// TIA Portal V19 export
DATA_BLOCK "DB_Prog_edit"   // DB800
{ S7_Optimized_Access := 'FALSE' }
// stored: AutoNumber false
   VAR RETAIN
      akt_edit_prog : Int;
      akt_Aufgabe_Prog : Int;
      old_Aufgabe_Prog : Int;   // Hilfsvariable um Programm in Aufgabestruktur zu kopieren
      resW : Int;
      resW_1 : Int;
      resD : DInt;
      Variante : USInt;   // 1=KSvl, 2=KSvr, 3=GOli, 4= GOre,5=KShl, 6=kshr, 7=LSv(BE1), 8= LSh(BE5)
      StandNr : USInt;
      GZ_Charge : DInt;
      Prog : Array[1..100] of Struct
         "Name" : String[100];
         Geometrie : USInt;   // 0=k.A., 1=KS, 2=LS, 3=GO
         ParaByte : USInt;   // .0=lgsm senken, .1=lgsm heben
         Faktor_ATZ : Real;
         resD : DInt;
         resW : Int;
         CM03_VorSpuel : Struct
            Expo : Time_Of_Day;
            Anfahren : Bool;
            res : Bool;
            res_1 : Bool;
            res_2 : Bool;
            res_3 : Bool;
            res_4 : Bool;
            res_5 : Bool;
            res_6 : Bool;
            resB : Byte;
            resW : Int;
            resD : DInt;
         END_STRUCT;
         CM01_VorAetz : Struct
            Expo : Time_Of_Day;
            Anfahren : Bool;
            res : Bool;
            res_1 : Bool;
            res_2 : Bool;
            res_3 : Bool;
            res_4 : Bool;
            res_5 : Bool;
            res_6 : Bool;
            Anzahl_Voraetz : Byte;
            resW : Int;
            resD : DInt;
         END_STRUCT;
         CM03_SpuelVorAetz : Struct
            Expo : Time_Of_Day;
            Anfahren : Bool;
            res : Bool;
            res_1 : Bool;
            res_2 : Bool;
            res_3 : Bool;
            res_4 : Bool;
            res_5 : Bool;
            res_6 : Bool;
            resB : Byte;
            resW : Int;
            resD : DInt;
         END_STRUCT;
         CM01_Aetzen : Struct
            Expo : Time_Of_Day;
            resD : DInt;
            resD_1 : DInt;
         END_STRUCT;
         CM03_Spl_1 : Struct
            Expo : Time_Of_Day;
            resD : DInt;
            resD_1 : DInt;
         END_STRUCT;
         CM04_Spl_2 : Struct
            Expo : Time_Of_Day;
            resD : DInt;
            resD_1 : DInt;
         END_STRUCT;
      END_STRUCT;
      Prog_Aufgabe : Struct
         Prog : Struct
            "Name" : String[100];
            Geometrie : USInt;   // 0=k.A., 1=KS, 2=LS, 3=GO
            ParaByte : USInt;   // .0=lgsm senken, .1=lgsm heben
            Faktor_ATZ : Real;
            resD : DInt;
            resW : Int;
            CM03_VorSpuel : Struct
               Expo : Time_Of_Day;
               Anfahren : Bool;
               res : Bool;
               res_1 : Bool;
               res_2 : Bool;
               res_3 : Bool;
               res_4 : Bool;
               res_5 : Bool;
               res_6 : Bool;
               resB : Byte;
               resW : Int;
               resD : DInt;
            END_STRUCT;
            CM01_VorAetz : Struct
               Expo : Time_Of_Day;
               Anfahren : Bool;
               res : Bool;
               res_1 : Bool;
               res_2 : Bool;
               res_3 : Bool;
               res_4 : Bool;
               res_5 : Bool;
               res_6 : Bool;
               Anzahl_Voraetz : Byte;
               resW : Int;
               resD : DInt;
            END_STRUCT;
            CM03_SpuelVorAetz : Struct
               Expo : Time_Of_Day;
               Anfahren : Bool;
               res : Bool;
               res_1 : Bool;
               res_2 : Bool;
               res_3 : Bool;
               res_4 : Bool;
               res_5 : Bool;
               res_6 : Bool;
               resB : Byte;
               resW : Int;
               resD : DInt;
            END_STRUCT;
            CM01_Aetzen : Struct
               Expo : Time_Of_Day;
               resD : DInt;
               resD_1 : DInt;
            END_STRUCT;
            CM03_Spl_1 : Struct
               Expo : Time_Of_Day;
               resD : DInt;
               resD_1 : DInt;
            END_STRUCT;
            CM04_Spl_2 : Struct
               Expo : Time_Of_Day;
               resD : DInt;
               resD_1 : DInt;
            END_STRUCT;
         END_STRUCT;
         Korb_Nr : Int;
      END_STRUCT;
   END_VAR
BEGIN
END_DATA_BLOCK
